{attribute 'qualified_only'}
{attribute 'to_string'}
TYPE BasinStateDisp :
(
	set_xMin	:= 0,
	set_xMax	:= 1,
	set_yMin	:= 2,
	set_yMax	:= 3
);
END_TYPE

(* stored: Version 1.1.0.1, ProductVersion 3.1.4026.12
   DUT BasinStateDisp: Id {055569c0-fd7d-4537-85de-6c5550a4465b} *)
